(* CODESYS project Projeto_Elevador.project

Project tree, tasks and I/O mapping:
  Device : CODESYS Control Win V3, 3S - Smart Software Solutions GmbH, order no. 305021, version 3.5.11.40
    application Application
      libraries: Standard, * (System)
      task MainTask (cyclic, interval t#20ms, priority 1) calls Main
      task Tarefa_Controle (cyclic, interval t#20ms, priority 1) calls Atende_Chamadas
      task Tarefa_Posicao (cyclic, interval t#20ms, priority 1) calls Posicao_Elevador
      global variables Var_GlobalList
      program Posicao_Elevador [ST]
      Symbols
      function block Aciona_Fins_de_Curso [ST]
      function block Atualiza_Mostradores_LCD [ST]
      program Main [SFC]: Andar_Destino, Chamada_Elevador, EMG_active, EMG_Desce_active, Init_active, Mov_Elevador_active, Fechando_Porta_active, Abrindo_Porta_active, Espera_Chamadas_active, Sobrecarga, Sobrecarga_active, Porta_Fechada, Porta_Aberta, EMG_Terreo_exit, Terreo, EMG_Terreo_active
      function block Fecha_Porta [ST]
      data type E_EstadoPorta
      function block Abre_Porta [ST]
      program Atende_Chamadas [ST]
*)

// Device/Application/E_EstadoPorta
{attribute 'qualified_only'}
{attribute 'strict'}
TYPE E_EstadoPorta :
(
    PORTA_ABERTA_ESPERANDO := 0,
    PORTA_FECHANDO         := 1,
    ESMAGAMENTO_DETECTADO  := 2,
    PORTA_FECHADA          := 3
);
END_TYPE

// Device/Application/Var_GlobalList
VAR_GLOBAL
    YY_T : BOOL;   // Sensor fim-de-curso ZIC_1 térreo (saida)
    YY_1 : BOOL;   // Sensor fim-de-curso ZIC_1 1      (saida)
    YY_2 : BOOL;   // Sensor fim-de-curso ZIC_1 2      (saida)
    YY_3 : BOOL;   // Sensor fim-de-curso ZIC_1 3      (saida)

    ZIC_1 : REAL;  // Sensor ultrassônico (saida)
    WIC_1 : INT;   // Célula de carga     (entrada)

    YY_ENT_SAI : BOOL;  // Sensor laser         (entrada)
    YY_ESMAG   : BOOL;  // Detector esmagamento (entrada)

    YY_IBT : BOOL;  // Botão interno T (entrada)
    YY_IB1 : BOOL;  // Botão interno 1 (entrada)
    YY_IB2 : BOOL;  // Botão interno 2 (entrada)
    YY_IB3 : BOOL;  // Botão interno 3 (entrada)

    YY_EBT : BOOL;  // Botão externo T (entrada)
    YY_EB1 : BOOL;  // Botão externo 1 (entrada)
    YY_EB2 : BOOL;  // Botão externo 2 (entrada)
    YY_EB3 : BOOL;  // Botão externo 3 (entrada)

    YY_EMG    : BOOL;  // Botão emergência (entrada)
    YY_REARME : BOOL;  // Chave rearme     (entrada)

    M_SOBE    : BOOL;  // Motor sobe          (saída)
    M_DESCE   : BOOL;  // Motor desce         (saída)
    VEL_MOTOR : REAL;  // Velocidade do motor (saída)
	
    M_ABRE_PORTA  : BOOL;  // Motor abre porta     (saída)
    M_FECHA_PORTA : BOOL;  // Motor fecha porta    (saída)
	YY_P_ABERTA   : BOOL;  // Sensor porta aberta  (saida)
	YY_P_FECHADA  : BOOL;  // Sensor porta fechada (saida)
	
    LD_IT : BOOL;   // LED interno T (saída)
    LD_I1 : BOOL;   // LED interno 1 (saída)
    LD_I2 : BOOL;   // LED interno 2 (saída)
    LD_I3 : BOOL;   // LED interno 3 (saída)

    LD_ET : BOOL;   // LED externo T (saída)
    LD_E1 : BOOL;   // LED externo 1 (saída)
    LD_E2 : BOOL;   // LED externo 2 (saída)
    LD_E3 : BOOL;   // LED externo 3 (saída)

    LD_PESO : BOOL;   // Lâmpada excesso peso (saída)

    LCD_I  : REAL;   // Mostrador LCD interno   (saída)
    LCD_T  : REAL;   // Mostrador LCD térreo    (saída)
    LCD_E1 : REAL;   // Mostrador LCD ZIC_1 1 (saída)
    LCD_E2 : REAL;   // Mostrador LCD ZIC_1 2 (saída)
    LCD_E3 : REAL;   // Mostrador LCD ZIC_1 3 (saída)

    BUZINA : BOOL;   // Buzina (saída)
	F_EMG  : BOOL;   // Flag para indicar estado de emergência
END_VAR

// Device/Application/Main
PROGRAM Main
VAR
	Func_Fecha_Porta : Fecha_Porta;
	Func_Abre_Porta  : Abre_Porta;
END_VAR

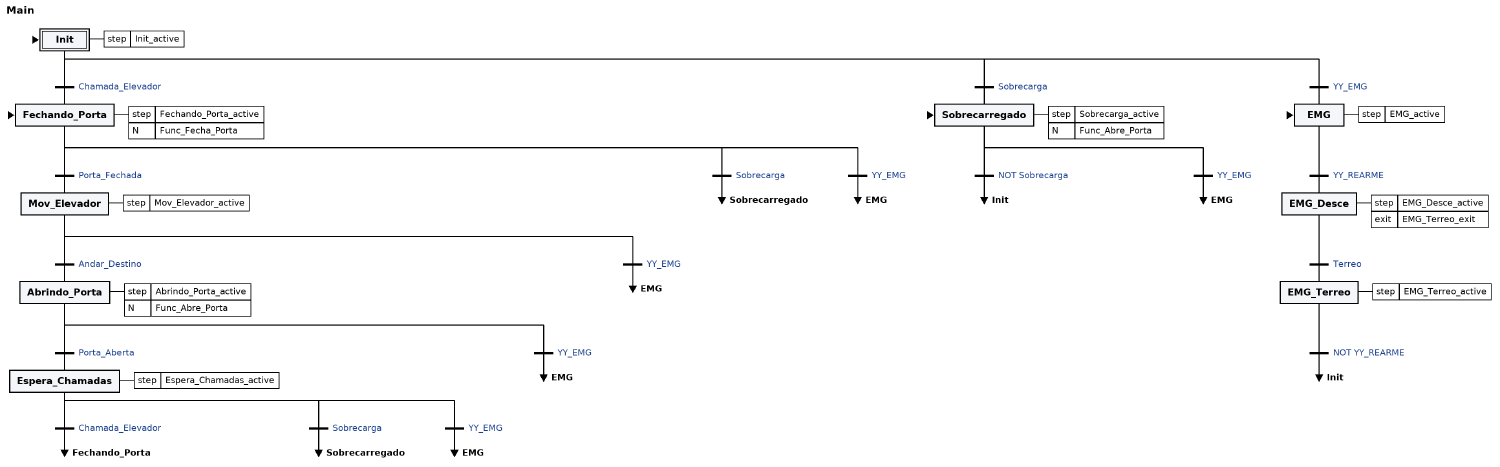
INITIAL_STEP Init:
    Init_active(N);  // step action
END_STEP
TRANSITION FROM Init TO Fechando_Porta
    := Chamada_Elevador;
END_TRANSITION
TRANSITION FROM Init TO Sobrecarregado
    := Sobrecarga;
END_TRANSITION
STEP Sobrecarregado:
    Sobrecarga_active(N);  // step action
    Func_Abre_Porta(N);
END_STEP
TRANSITION FROM Sobrecarregado TO Init
    := NOT Sobrecarga;
END_TRANSITION
TRANSITION FROM Sobrecarregado TO EMG
    := YY_EMG;
END_TRANSITION
STEP Fechando_Porta:
    Fechando_Porta_active(N);  // step action
    Func_Fecha_Porta(N);
END_STEP
TRANSITION FROM Fechando_Porta TO Mov_Elevador
    := Porta_Fechada;
END_TRANSITION
TRANSITION FROM Fechando_Porta TO Sobrecarregado
    := Sobrecarga;
END_TRANSITION
TRANSITION FROM Fechando_Porta TO EMG
    := YY_EMG;
END_TRANSITION
TRANSITION FROM Init TO EMG
    := YY_EMG;
END_TRANSITION
STEP EMG:
    EMG_active(N);  // step action
END_STEP
TRANSITION FROM EMG TO EMG_Desce
    := YY_REARME;
END_TRANSITION
STEP EMG_Desce:
    EMG_Desce_active(N);  // step action
    EMG_Terreo_exit(P0);  // exit action
END_STEP
TRANSITION FROM EMG_Desce TO EMG_Terreo
    := Terreo;
END_TRANSITION
STEP EMG_Terreo:
    EMG_Terreo_active(N);  // step action
END_STEP
TRANSITION FROM EMG_Terreo TO Init
    := NOT YY_REARME;
END_TRANSITION
STEP Mov_Elevador:
    Mov_Elevador_active(N);  // step action
END_STEP
TRANSITION FROM Mov_Elevador TO Abrindo_Porta
    := Andar_Destino;
END_TRANSITION
TRANSITION FROM Mov_Elevador TO EMG
    := YY_EMG;
END_TRANSITION
STEP Abrindo_Porta:
    Abrindo_Porta_active(N);  // step action
    Func_Abre_Porta(N);
END_STEP
TRANSITION FROM Abrindo_Porta TO Espera_Chamadas
    := Porta_Aberta;
END_TRANSITION
STEP Espera_Chamadas:
    Espera_Chamadas_active(N);  // step action
END_STEP
TRANSITION FROM Espera_Chamadas TO Fechando_Porta
    := Chamada_Elevador;
END_TRANSITION
TRANSITION FROM Espera_Chamadas TO Sobrecarregado
    := Sobrecarga;
END_TRANSITION
TRANSITION FROM Espera_Chamadas TO EMG
    := YY_EMG;
END_TRANSITION
TRANSITION FROM Abrindo_Porta TO EMG
    := YY_EMG;
END_TRANSITION

TRANSITION Andar_Destino:
// Elevador chegou no andar de destino
(
(Atende_Chamadas.AndarDestino = 0 AND YY_T) AND (NOT YY_EMG) OR  // Chegou no Térreo
(Atende_Chamadas.AndarDestino = 1 AND YY_1) AND (NOT YY_EMG) OR  // Chegou no 1º Andar
(Atende_Chamadas.AndarDestino = 2 AND YY_2) AND (NOT YY_EMG) OR  // Chegou no 2º Andar
(Atende_Chamadas.AndarDestino = 3 AND YY_3) AND (NOT YY_EMG)     // Chegou no 3º Andar
) AND NOT YY_EMG
END_TRANSITION

TRANSITION Chamada_Elevador:
Atende_Chamadas.NumChamadas > 0 AND NOT YY_EMG AND NOT Sobrecarga
END_TRANSITION

ACTION EMG_active:
// Aciona Buzina
BUZINA := TRUE;

// Estado de emergência
F_EMG := TRUE;

// Garante que o elevador nao se move
Posicao_Elevador.Movimenta := FALSE;
END_ACTION

ACTION EMG_Desce_active:
// Aciona Buzina
BUZINA := TRUE;

// Estado de emergência
F_EMG := TRUE;

// Elevador desce para o Térreo
Posicao_Elevador.Movimenta := TRUE;
END_ACTION

ACTION Init_active:
// Elevador no térreo
ZIC_1 := 0;

// Porta aberta
YY_P_ABERTA  := TRUE;
YY_P_FECHADA := FALSE;

// Motores de abertura e fechamento da porta desligados
M_ABRE_PORTA  := FALSE;
M_FECHA_PORTA := FALSE;

// Motores de sobida e descida desligados
M_SOBE    := 0;
M_DESCE   := 0;
VEL_MOTOR := 0;

// Elevador não se movimenta
Posicao_Elevador.Movimenta := FALSE;

// Sem emergência
F_EMG := FALSE;
Atende_Chamadas.Zera_Chamadas := FALSE;
END_ACTION

ACTION Mov_Elevador_active:
// Elevador pode se movimentar
Posicao_Elevador.Movimenta := TRUE;
END_ACTION

ACTION Fechando_Porta_active:
// Elevador não se movimenta
Posicao_Elevador.Movimenta := FALSE;
END_ACTION

ACTION Abrindo_Porta_active:
// Elevador não se movimenta
Posicao_Elevador.Movimenta := FALSE;
END_ACTION

ACTION Espera_Chamadas_active:
// Elevador não se movimenta
Posicao_Elevador.Movimenta := FALSE;

// Desliga motores
M_ABRE_PORTA  := FALSE;
M_FECHA_PORTA := FALSE;
VEL_MOTOR     := 0;

// Indica o andar atual ao elevador
Posicao_Elevador.UltimoAndar := Atende_Chamadas.PosicaoAtual;
END_ACTION

TRANSITION Sobrecarga:
WIC_1 > 700 AND NOT YY_EMG
END_TRANSITION

ACTION Sobrecarga_active:
// Elevador não se movimenta
Posicao_Elevador.Movimenta := FALSE;

// Acende LED de sobrecarga
LD_PESO := TRUE;
END_ACTION

TRANSITION Porta_Fechada:
YY_P_FECHADA AND NOT YY_EMG AND NOT Sobrecarga
END_TRANSITION

TRANSITION Porta_Aberta:
YY_P_ABERTA AND NOT YY_EMG
END_TRANSITION

ACTION EMG_Terreo_exit:
// Zera todas as chamadas ao sair do estado
Atende_Chamadas.Zera_Chamadas := TRUE;
END_ACTION

TRANSITION Terreo:
ZIC_1 < 0.1
END_TRANSITION

ACTION EMG_Terreo_active:
// Aciona Buzina
BUZINA := TRUE;

// Estado de emergência
F_EMG := TRUE;

// Para ao chegar ao Térreo
Posicao_Elevador.Movimenta := FALSE;

// Zera todas as chamadas
Atende_Chamadas.Zera_Chamadas := TRUE;
END_ACTION

END_PROGRAM

// Device/Application/Fecha_Porta
(*   
	Function Block: Fecha_Porta
	
 	Descrição:
	
	Este Function Block implementa uma máquina de estados  para gerenciar o fechamento
	da porta do elevador. Os estados são:
	1. Espera de passageiros;
	2. Fechamento da porta; 
	3. Detecção de  esmagamento com reabertura automática; 
	4. Porta fechada.
	
	O estado da porta (aberta, fechada ou em movimento) é alterado em cada estado
*)

FUNCTION_BLOCK Fecha_Porta
VAR_INPUT
END_VAR
VAR_OUTPUT
END_VAR
VAR
	// Possiveis estados da porta do elevador
    estadoPorta : E_EstadoPorta := E_EstadoPorta.PORTA_ABERTA_ESPERANDO; 
	
	START : BOOL := TRUE;  // Variavel de controle usada para começar sempre do Estado PORTA_ABERTA_ESPERANDO
	
	TMR_Espera_Passageiro : TON; // Temporizador de 5s para aguardar passageiro
    TMR_Acao_Motor 	      : TON; // Temporizador de 3s para manter motores da porta acionados
END_VAR

// Garante que o CASE volta para o estado de PORTA_ABERTA_ESPERANDO após a primeira iteração
IF YY_P_ABERTA AND START THEN 
	estadoPorta := E_EstadoPorta.PORTA_ABERTA_ESPERANDO;
END_IF;

CASE estadoPorta OF
	
	// Estado 1: Porta aberta e esperando passageiros
    E_EstadoPorta.PORTA_ABERTA_ESPERANDO:
		START := FALSE;
		
        // Garante que os motores da porta estão desligados
        M_ABRE_PORTA  := FALSE;
        M_FECHA_PORTA := FALSE;
		
		// Porta aberta
		YY_P_ABERTA  := TRUE;
		YY_P_FECHADA := FALSE;

        // Espera 5 segundos consecutivos sem ninguém entrar no elevador
        TMR_Espera_Passageiro(
            IN:= NOT YY_ENT_SAI,
            PT:= T#5S
        );

        // Se o tempo de 5s se esgotou sem detecção de passageiros, muda para o Estado PORTA_FECHANDO.
        IF TMR_Espera_Passageiro.Q THEN
            estadoPorta :=   E_EstadoPorta.PORTA_FECHANDO;
            TMR_Espera_Passageiro(IN:= FALSE); // Reseta o timer de espera para o próximo uso.
        END_IF;

	
	// Estado 2: Porta começa a se fechar
      E_EstadoPorta.PORTA_FECHANDO:
		// Porta fechando
		YY_P_ABERTA  := FALSE;
		YY_P_FECHADA := FALSE;
	
        // Se for o sensor de esmagamento for ativado, a porta deve reabrir
        IF YY_ESMAG THEN
            estadoPorta :=   E_EstadoPorta.ESMAGAMENTO_DETECTADO;
            TMR_Acao_Motor(IN:= FALSE); // Interrompe e reseta o timer de fechamento
            M_FECHA_PORTA := FALSE;     // Garante que o motor de fechar pare

        ELSE
            // Se não há esmagamento, liga o motor para fechar a porta
            M_FECHA_PORTA := TRUE;
            M_ABRE_PORTA  := FALSE;

            // Ativa o timer de ação do motor por 3 segundos
            TMR_Acao_Motor(IN:= TRUE, PT:= T#3S);

            // Passaram-se 3 segundos, porta fechada
            IF TMR_Acao_Motor.Q THEN
				// Porta fechada
				YY_P_ABERTA  := FALSE;
				YY_P_FECHADA := TRUE;
				
                estadoPorta :=   E_EstadoPorta.PORTA_FECHADA;
                TMR_Acao_Motor(IN:= FALSE); // Reseta o timer.
            END_IF;
        END_IF;

	// Estado 3: Sensor detecta esmagamento
      E_EstadoPorta.ESMAGAMENTO_DETECTADO:
		// Porta abrindo
		YY_P_ABERTA  := FALSE;
		YY_P_FECHADA := FALSE;
		
        // Liga o motor para abrir a porta.
        M_ABRE_PORTA  := TRUE;
        M_FECHA_PORTA := FALSE;

        // Ativa o timer de ação do motor por 3 segundos.
        TMR_Acao_Motor(IN:= TRUE, PT:= T#3S);

        // Quando o tempo de 3s acabar, a porta é considerada aberta e o ciclo reinicia.
        IF TMR_Acao_Motor.Q THEN
            estadoPorta :=   E_EstadoPorta.PORTA_ABERTA_ESPERANDO; // Volta a esperar passageiros.
            TMR_Acao_Motor(IN:= FALSE); // Reseta o timer.
        END_IF;

	
	// Estado 4: Porta fechada
      E_EstadoPorta.PORTA_FECHADA:
        // Garante que todos os motores estão desligados.
        M_ABRE_PORTA  := FALSE;
        M_FECHA_PORTA := FALSE;
		
		// Porta fechada
		YY_P_ABERTA  := FALSE;
		START 		 := TRUE;
		YY_P_FECHADA := TRUE;
END_CASE;

END_FUNCTION_BLOCK

// Device/Application/Abre_Porta
FUNCTION_BLOCK Abre_Porta
VAR
    TON_Abre : TON;
END_VAR

// Garante que a porta não está fechada
M_FECHA_PORTA := FALSE;
YY_P_FECHADA  := FALSE;

// Logica para temporizador do motor abre porta
IF NOT YY_P_ABERTA THEN
    M_ABRE_PORTA  := TRUE;
    TON_Abre(IN := TRUE, PT := T#3S);
ELSE
    M_ABRE_PORTA  := FALSE;
    TON_Abre(IN := FALSE, PT := T#3S);
END_IF;

// Abre a porta
IF TON_Abre.Q THEN
    YY_P_ABERTA := TRUE;
END_IF;

END_FUNCTION_BLOCK

// Device/Application/Atende_Chamadas
PROGRAM Atende_Chamadas
VAR_INPUT
	Zera_Chamadas: BOOL;  // Zera todas as chamadas do elevador
END_VAR
VAR_OUTPUT
	AndarDestino : INT := -1;  // Próximo andar a ser atendido
	NumChamadas  : INT := 0;   // Quantidade de chamadas registradas
	
END_VAR
VAR
	NovaChamada  : BOOL;                                // Novo andar chamado
	AndarChamado : INT;                                 // 0 -> Térreo; 1 -> 1º Andar; 2 -> 2º Andar; 3 -> 3º Andar
	Chamadas     : ARRAY[0..3] OF INT := [0, 0, 0, 0];  // Vetor de chamadas de andares.
														// Chamadas[n] = 1 -> Há chamada para o andar n
														// Chamadas[m] = 0 -> Não há chamada para o andar n

    PosicaoAtual : INT := 0;  // Andar atual do elevador
	UltimoAndar  : INT := 0;  // Ultimo Andar pelo qual o elevador passou
	Direcao      : INT := 1;  // 1 -> Subindo, -1 -> Descendo
END_VAR

IF NOT F_EMG AND NOT Zera_Chamadas THEN
	// Verifica qual o andar chamado
	IF (YY_IBT OR YY_EBT) AND PosicaoAtual <> 0 THEN
		AndarChamado := 0;
		NovaChamada  := TRUE;
	ELSIF (YY_IB1 OR YY_EB1) AND PosicaoAtual <> 1 THEN
		AndarChamado := 1;
		NovaChamada  := TRUE;
	ELSIF (YY_IB2 OR YY_EB2)  AND PosicaoAtual <> 2 THEN
		AndarChamado := 2;
		NovaChamada  := TRUE;
	ELSIF (YY_IB3 OR YY_EB3) AND PosicaoAtual <> 3 THEN
		AndarChamado := 3;
		NovaChamada  := TRUE;
	END_IF
	
	// Adiciona novas chamadas
	IF NovaChamada THEN
		// Checa se o andar já foi chamado
		IF Chamadas[AndarChamado] = 1 THEN 
			// Não faz nada se o andar já foi chamado
			NovaChamada  := FALSE;
		ELSE
			// Preenche Chamadas[] na posicao correta 
			IF AndarChamado = 0 THEN
				Chamadas[0] := 1;
				NovaChamada  := FALSE;
			ELSIF AndarChamado = 1 THEN
				Chamadas[1] := 1;
				NovaChamada  := FALSE;					
			ELSIF AndarChamado = 2 THEN
				Chamadas[2] := 1;
				NovaChamada  := FALSE;	
			ELSIF AndarChamado = 3 THEN
				Chamadas[3] := 1;
				NovaChamada  := FALSE;
			END_IF
		END_IF
	END_IF
	
	// Conta chamadas
	NumChamadas := 0;
	IF Chamadas[0] = 1 THEN
		NumChamadas := NumChamadas +1; 
	END_IF
	IF Chamadas[1] = 1 THEN
		NumChamadas := NumChamadas +1; 
	END_IF
	IF Chamadas[2] = 1 THEN
		NumChamadas := NumChamadas +1; 
	END_IF
	IF Chamadas[3] = 1 THEN
		NumChamadas := NumChamadas +1; 
	END_IF
	
	// Atende Chamadas
	IF NumChamadas > 0 THEN
	
		 // Caso elevador SUBINDO
		IF Direcao = 1 THEN
			IF PosicaoAtual = 0 OR UltimoAndar = 0 THEN  // Elevador no TERREO
				IF Chamadas[1] = 1 THEN // Chamada no 1º Andar
					AndarDestino := 1;  
				ELSIF Chamadas[2] = 1 THEN  // Chamada no 2º Andar
					AndarDestino := 2;
				ELSIF Chamadas[3] = 1 THEN  // Chamada no 3º Andar
					AndarDestino := 3;
				END_IF
			ELSIF PosicaoAtual = 1 OR UltimoAndar = 1 THEN  // Elevador no 1º ANDAR
				IF Chamadas[2] = 1 THEN  // Chamada no 2º Andar
					AndarDestino := 2;
				ELSIF Chamadas[3] = 1 THEN  // Chamada no 3º Andar
					AndarDestino := 3;
				ELSE
					Direcao := -1;  // Muda direcao do elevador
				END_IF
			ELSIF PosicaoAtual = 2 OR UltimoAndar = 2 THEN  // Elevador no 2º ANDAR
				IF Chamadas[3] = 1 THEN  // Chamada no 3º Andar
					AndarDestino := 3;
				ELSE
					Direcao := -1;  // Muda direcao do elevador
				END_IF
			ELSIF PosicaoAtual = 3 OR UltimoAndar = 3 THEN  // Elevador no 3º ANDAR
				Direcao := -1;      // Muda direcao do elevador
			END_IF
		END_IF
		
		 // Caso elevador DESCENDO
		IF Direcao = -1 THEN
			IF PosicaoAtual = 3 OR UltimoAndar = 3 THEN  // Elevador no 3º Andar
				IF Chamadas[2] = 1 THEN // Chamada no 2º Andar
					AndarDestino := 2;  
				ELSIF Chamadas[1] = 1 THEN  // Chamada no 1º Andar
					AndarDestino := 1;
				ELSIF Chamadas[0] = 1 THEN  // Chamada no TERREO
					AndarDestino := 0;
				END_IF
			ELSIF PosicaoAtual = 2 OR UltimoAndar = 2 THEN  // Elevador no 2º Andar
				IF Chamadas[1] = 1 THEN  // Chamada no 1º Andar
					AndarDestino := 1;
				ELSIF Chamadas[0] = 1 THEN  // Chamada no TERREO
					AndarDestino := 0;
				ELSE
					Direcao := 1;  // Muda direcao do elevador
				END_IF
			ELSIF PosicaoAtual = 1 OR UltimoAndar = 1 THEN  // Elevador no 1º Andar
				IF Chamadas[0] = 1 THEN  // Chamada no TERREO
					AndarDestino := 0;
				ELSE 
					Direcao := 1;  // Muda direcao do elevador
				END_IF
			ELSIF PosicaoAtual = 0 OR UltimoAndar = 0 THEN  // Elevador no 3º Andar
				Direcao := 1;      // Muda direcao do elevador
			END_IF
		END_IF
	
	END_IF
	
	// Atualiza posição atual
	IF YY_T THEN
		PosicaoAtual := 0;   // Térreo
		UltimoAndar  := 0;
	ELSIF YY_1 THEN
		PosicaoAtual := 1;   // 1º Andar
		UltimoAndar  := 1;
	ELSIF YY_2 THEN
		PosicaoAtual := 2;   // 2º Andar
		UltimoAndar  := 2;
	ELSIF YY_3 THEN
		PosicaoAtual := 3;   // 3º Andar
		UltimoAndar  := 3;
	ELSE 
		PosicaoAtual := -1;  // Elevador em trânsito
	END_IF
	
	// Chegou ao destino
	IF PosicaoAtual = AndarDestino THEN
		Chamadas[PosicaoAtual] := 0;
	END_IF
	
	// Acende e apaga botões
	IF Chamadas[0] = 1 THEN  // Térreo
		LD_IT := TRUE;
		LD_ET := TRUE;
	ELSE
		LD_IT := FALSE;
		LD_ET := FALSE;
	END_IF
	IF Chamadas[1] = 1 THEN  // 1º Andar
		LD_I1 := TRUE;
		LD_E1 := TRUE;
	ELSE
		LD_I1 := FALSE;
		LD_E1 := FALSE;
	END_IF
	IF Chamadas[2] = 1 THEN  // 2º Andar
		LD_I2 := TRUE;
		LD_E2 := TRUE;
	ELSE
		LD_I2 := FALSE;
		LD_E2 := FALSE;
	END_IF
	IF Chamadas[3] = 1 THEN  // 3º Andar
		LD_I3 := TRUE;
		LD_E3 := TRUE;
	ELSE
		LD_I3 := FALSE;
		LD_E3 := FALSE;
	END_IF
	
ELSIF F_EMG AND NOT Zera_Chamadas THEN // Emergencia. Reiniciar estado do elevador
	// Elevador deve ir para o Térreo
	AndarChamado := 0;
	NovaChamada  := TRUE;
	
	// Zera as chamadas, com excecao do Terreo
	Chamadas[0] := 1;
	Chamadas[1] := 0;
	Chamadas[2] := 0;
	Chamadas[3] := 0;
	NumChamadas  := 1;
	
	// Desce para o Térreo
	AndarDestino := 0;
	Direcao   := -1;

ELSIF Zera_Chamadas THEN
	NovaChamada  := FALSE;
	AndarChamado := 0;

	Chamadas[0] := 0;
	Chamadas[1] := 0;
	Chamadas[2] := 0;
	Chamadas[3] := 0;
	
    PosicaoAtual := 0;
	UltimoAndar  := 0;
	Direcao      := 1;

END_IF

END_PROGRAM

// Device/Application/Posicao_Elevador
PROGRAM Posicao_Elevador
VAR CONSTANT
	Velocidade_Baixa : REAL := 0.00333;  // Equivale a 10m/min
	Velocidade_Alta  : REAL := 0.01;     // Equivale a 30m/min
END_VAR
VAR_INPUT
	Movimenta   : BOOL := FALSE;  // Usado para mover ou nao o elevador
	UltimoAndar : REAL := 0;      // Andar do qual o elevador partiu por ultimo
END_VAR
VAR
	Velocidade : REAL;	

	Sobe  : BOOL := TRUE;
	Desce : BOOL := FALSE;
		
	Fins_de_Curso : Aciona_Fins_de_Curso;     // Função para acionar e desativar os fins de curso em cada andar.
	LCDs          : Atualiza_Mostradores_LCD; // Função para atualizar os mostradores LCDs

END_VAR

// Verifica se o elevador deve subir ou descer
IF Atende_Chamadas.Direcao = 1 THEN 
	Sobe := TRUE; 
	Desce := FALSE;
ELSIF Atende_Chamadas.Direcao = -1 THEN
	Sobe := FALSE; 
	Desce := TRUE;
END_IF

// Controla a velocidade do elevador
IF Sobe THEN
	IF ZIC_1 < (UltimoAndar * 4 + 1) OR                // Elevador há menos de 1 metro do andar de partida
	   ZIC_1 > (Atende_Chamadas.AndarDestino * 4 - 1)  // Elevador há menos de 1 metro do andar de chegada
	THEN             
		Velocidade := Velocidade_Baixa;
		VEL_MOTOR  := 10;	
	ELSE
		Velocidade := Velocidade_Alta;
		VEL_MOTOR  := 30;
	END_IF
ELSIF Desce THEN
	IF ZIC_1 > (UltimoAndar * 4 - 1) OR                // Elevador há menos de 1 metro do andar de partida
	   ZIC_1 < (Atende_Chamadas.AndarDestino * 4 + 1)  // Elevador há menos de 1 metro do andar de chegada
	THEN
		Velocidade := Velocidade_Baixa;
		VEL_MOTOR  := 10;
	ELSE
		Velocidade := Velocidade_Alta;
		VEL_MOTOR  := 30;
	END_IF
END_IF

// Controla posição do Elevador
IF NOT Movimenta THEN
	M_SOBE    := FALSE;
	M_DESCE   := FALSE;
	VEL_MOTOR := 0;
	
ELSIF Sobe AND Movimenta THEN 
	ZIC_1 := ZIC_1 + Velocidade;
	M_SOBE  := TRUE;
	M_DESCE := FALSE;
	
ELSIF Desce AND Movimenta THEN 
	ZIC_1 := ZIC_1 - Velocidade;
	M_SOBE  := FALSE;
	M_DESCE := TRUE;
END_IF

// Aciona ou desativa os fins de curso de cada andar
Fins_de_Curso(Posicao := ZIC_1);

// Atualiza os Mostradores LDC
LCDs();

END_PROGRAM

// Device/Application/Aciona_Fins_de_Curso
(*   
	Function Block: Aciona_Fins_de_Curso
	
 	Descrição:
  	Este Function Block lê a atual posição do elevador e aciona o fim de curso correspondente
	ao seu andar, desativando todos os outros. Se o elevador não estiver parado em nenhum andar,
	todos os fins de curso são desativados
*)

FUNCTION_BLOCK Aciona_Fins_de_Curso
VAR_INPUT
	Posicao : REAL;  // Posição do vertical do elevador (m)
END_VAR
VAR_OUTPUT
END_VAR
VAR
END_VAR

// Elevador no Térreo
IF ZIC_1 >= -0.1 AND ZIC_1 <= 0.1 THEN
    YY_T := TRUE;
    YY_1 := FALSE;
    YY_2 := FALSE;
    YY_3 := FALSE;

// Elevador no 1º Andar
ELSIF ZIC_1 >= 3.9 AND ZIC_1 <= 4.1 THEN
    YY_T := FALSE;
    YY_1 := TRUE;
    YY_2 := FALSE;
    YY_3 := FALSE;

// Elevador no 2º Andar
ELSIF ZIC_1 >= 7.9 AND ZIC_1 <= 8.1 THEN
    YY_T := FALSE;
    YY_1 := FALSE;
    YY_2 := TRUE;
    YY_3 := FALSE;

// Elevador no 3º Andar
ELSIF ZIC_1 >= 11.9 AND ZIC_1 <= 12.1 THEN
    YY_T := FALSE;
    YY_1 := FALSE;
    YY_2 := FALSE;
    YY_3 := TRUE;

// Elevador em trânsito
ELSE
    YY_T := FALSE;
    YY_1 := FALSE;
    YY_2 := FALSE;
    YY_3 := FALSE;
END_IF;

END_FUNCTION_BLOCK

// Device/Application/Atualiza_Mostradores_LCD
(*   
	Function Block: Mostradores_LCD
	
 	Descrição:
  	Este Function Block exibe o andar no qual está localizado o elevador. Se o elevador 
	estiver entre andares, será exibido o último andar.
*)

FUNCTION_BLOCK Atualiza_Mostradores_LCD
VAR_INPUT
END_VAR
VAR_OUTPUT
END_VAR
VAR
END_VAR

// Elevador no Térreo
IF YY_T = TRUE THEN
	LCD_I  := 0;
    LCD_T  := 0;
    LCD_E1 := 0;
    LCD_E2 := 0;
    LCD_E3 := 0;

// Elevador no 1º Andar
ELSIF YY_1 = TRUE THEN
	LCD_I  := 1;
    LCD_T  := 1;
    LCD_E1 := 1;
    LCD_E2 := 1;
    LCD_E3 := 1;
	
// Elevador no 2º Andar
ELSIF YY_2 = TRUE THEN
	LCD_I  := 2;
    LCD_T  := 2;
    LCD_E1 := 2;
    LCD_E2 := 2;
    LCD_E3 := 2;

// Elevador no 3º Andar
ELSIF YY_3 = TRUE THEN
	LCD_I  := 3;
    LCD_T  := 3;
    LCD_E1 := 3;
    LCD_E2 := 3;
    LCD_E3 := 3;

END_IF

END_FUNCTION_BLOCK
